FUNCTION_BLOCK CmdAndIlcked (* Basic Function Block Type *)
  (* Standard: 61499-2 *)
  (* Version 0.0, 7/31/2026, Schneider Electric, Template *)
  PACKAGE SE.Nereda;
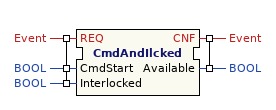
  EVENT_INPUT
    REQ WITH CmdStart, Interlocked; (* Normal Execution Request *)
  END_EVENT
  EVENT_OUTPUT
    CNF WITH Available; (* Execution Confirmation *)
  END_EVENT
  VAR_INPUT
    CmdStart : BOOL;
    Interlocked : BOOL;
  END_VAR
  VAR_OUTPUT
    Available : BOOL;
  END_VAR
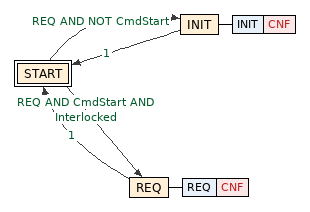
  EC_STATES
    START; (* Initial State *)
    INIT : INIT -> CNF; (* Initialization *)
    REQ : REQ -> CNF; (* Normal execution *)
  END_STATES
  EC_TRANSITIONS
    START TO INIT := REQ AND NOT CmdStart;
    INIT TO START := 1;
    START TO REQ := REQ AND CmdStart AND Interlocked;
    REQ TO START := 1;
  END_TRANSITIONS
  ALGORITHM INIT IN ST: (* Initialization algorithm *)
;
Available := TRUE;
  END_ALGORITHM
  ALGORITHM REQ IN ST: (* Normally executed algorithm *)
;
Available := FALSE;
  END_ALGORITHM
END_FUNCTION_BLOCK
